{attribute 'linkalways'} 
{attribute 'no_explicit_call' := 'This FB is a CLASS and must be accessed using methods or properties'}
{attribute 'enable_dynamic_creation'}
FUNCTION_BLOCK FINAL OR_DWORD EXTENDS Node
VAR
	in1 : _DWORD(0);
	in2 : _DWORD(0);
	out : _DWORD(0);
END_VAR

METHOD PUBLIC Clone : I_Node
VAR
	pNode : POINTER TO OR_DWORD;
END_VAR
pNode := __NEW(OR_DWORD);
Clone := pNode^;
END_METHOD

METHOD FB_init : BOOL
VAR_INPUT
	bInitRetains : BOOL; // if TRUE, the retain variables are initialized (warm start / cold start)
	bInCopyCode : BOOL;  // if TRUE, the instance afterwards gets moved into the copy code (online change)
END_VAR
AddInput('in1',THIS^.in1);
AddInput('in2',THIS^.in2);
AddOutput('out', THIS^.out);
END_METHOD

METHOD PROTECTED OnExecute
VAR
END_VAR
out.Value := in1.Value OR in2.Value;
END_METHOD

END_FUNCTION_BLOCK

(* stored: Version 1.1.0.1, ProductVersion 3.1.4024.15
   POU OR_DWORD: Id {86f1655a-4a65-4a99-a8e4-828ea6d15a1b}, SpecialFunc None
   Folder Constructor: Id {64dbd8ba-35c3-4870-9324-1f259dc17925}
   Method Clone: Id {3fbab1d4-79cb-4307-a116-cd8d30e2ddcd}
   Method FB_init: Id {583c9483-95bc-4272-b9dd-a38fc01fb461}
   Method OnExecute: Id {0dd2a5f8-ef0d-4b97-9a6f-c4379e7e2434} *)
